// TIA Portal V17 export
// export: Created 2025-03-07T09:16:19.2612714Z, ExportSetting WithDefaults, DisplayName Totally Integrated Automation Portal, DisplayVersion V17 Update 8, DisplayName TIA Portal Openness, DisplayVersion V17 Update 8, DisplayName TIA Portal Version Control Interface, DisplayVersion V17, DisplayName SINAMICS Startdrive Advanced, DisplayVersion V17 SP2, DisplayName SINAMICS Startdrive G110M, G120, G120C, G120D, G120P, G115D, DisplayVersion V17 SP2, DisplayName SINAMICS Startdrive G130, G150, S120, S150, SINAMICS MV, S210, DisplayVersion V17 SP2, DisplayName STEP 7 Professional, DisplayVersion V17 Update 8, DisplayName SINUMERIK ONE STEP 7 Toolbox, DisplayVersion V17 Update 12, DisplayName SINUMERIK 840D sl STEP 7 Toolbox, DisplayVersion V17 Update 12, DisplayName STEP 7 Safety, DisplayVersion V17 Update 6, DisplayName WinCC Advanced, DisplayVersion V17 Update 8
DATA_BLOCK "LBP_InternalDB1020"   // DB1020
TITLE = Internal DB for basic program / DB interno para el programa básico / Interner DB für Grundprogramm
{ DB_Accessible_From_OPC_UA := 'FALSE' }
// DB only for internal use in the basic program / DB solo para uso interno en el programa básico / DB nur zur internen Verwendung im Grundprogramm
// stored: AutoNumber false, DBAccessibleFromOPCUA false, DBAccessibleFromWebserver true, InstanceOfName LBP_InternalFB1020, InstanceOfType FB
"LBP_InternalFB1020"
   // VAR_INPUT
   //    IN1 : UDInt;
   //    IN2 : UDInt;
   //    IN3 : Word;
   //    IN4 : Variant;
   //    IN5 : Variant;
   //    IN6 : Variant;
   //    IN7 : Variant;
   //    IN8 : Variant;
   //    IN9 : Variant;
   //    IN10 : Variant;
   //    IN11 : Variant;
   //    IN12 : Variant;
   // END_VAR
   // VAR_OUTPUT
   //    OUT1 : Bool;
   //    OUT2 : DWord;
   //    OUT3 : UInt;
   // END_VAR
   // VAR
   //    LBP_AlarmType_ErrMsg { S7_SetPoint := 'True'} : Diag_Alarm;
   //    LBP_AlarmType_OpMsg { S7_SetPoint := 'True'} : Diag_Alarm;
   //    LBP_AlarmType_InfoMsg { S7_SetPoint := 'True'} : Diag_Alarm;
   //    LBP_DB2AlarmType_ErrMsg { S7_SetPoint := 'True'} : Diag_Alarm;
   //    LBP_DB2AlarmType_OpMsg { S7_SetPoint := 'True'} : Diag_Alarm;
   //    LBP_DB2AlarmType_InfoMsg { S7_SetPoint := 'True'} : Diag_Alarm;
   //    LBP_UserAlarmType_ErrMsg { S7_SetPoint := 'True'} : Diag_Alarm;
   //    LBP_UserAlarmType_OpMsg { S7_SetPoint := 'True'} : Diag_Alarm;
   //    LBP_UserAlarmType_InfoMsg { S7_SetPoint := 'True'} : Diag_Alarm;
   //    LBP_UserAlarmType_AckMsg { S7_SetPoint := 'True'} : Diag_Alarm;
   //    s_strct_DB2AddressLastCycle : Struct
   //       LwByteAddress : DInt;
   //       LwBitAddress : DInt;
   //    END_STRUCT;
   //    s_DB2_MaxScanByteUser : DInt;
   //    s_DB7_Params : Struct
   //       MaxAxis : Int;
   //       MaxChan : Int;
   //       MsgUser : Int;
   //       ExtendChanAxMsg : Bool;
   //       ActivChan : Array[1..10] of Bool;
   //       ActivAxis : Array[1..31] of Bool;
   //    END_STRUCT;
   //    s_firstScanFinished : Bool;
   //    s_FC10_Quit : Struct
   //       QuitEdge : Bool;
   //       LwByteAddress : DInt;
   //       DB2ScanFinished : Bool;
   //    END_STRUCT;
   //    s_CounterActiveDB2Alarms : UInt;
   //    s_FC10_ToUserIf_OLD : Bool;
   // END_VAR
BEGIN
END_DATA_BLOCK
